// TwinCAT 3 PLC project PLC3
// ProgramVersion: 3.1.4022.3
// libraries:
//   Tc2_Standard, * (Beckhoff Automation GmbH)
//   Tc2_System, * (Beckhoff Automation GmbH)
//   Tc3_Module, * (Beckhoff Automation GmbH)
// project tree:
//   DUTs/ Drinks.TcDUT (not stored), States.TcDUT (not stored)
//   / GlobalTextList.TcGTLO (not stored), PlcTask.TcTTO (not stored), Visualization Manager.TcVMO (not stored)
//   GVLs/ GVL_IO.TcGVL
//   POUs/ FindFree.TcPOU, MAIN.TcPOU, MoveArm.TcPOU, CountFreeSpaces.TcPOU (not stored)
// real-time tasks:
//   TASK PlcTask: cycle T#10ms, priority 20, ADS port 350
// I/O:
//   DEVICE Device 1 (EtherCAT), AmsNetId 5.17.58.102.2.1
//     Term 1 (EK1200) [EK1200-5000 EtherCAT Power supply (2A E-Bus)]
//       Term 2 (EK1110) [EK1110 EtherCAT extension]
//     Term 3 (EK1100) [EK1100 EtherCAT Coupler (2A E-Bus)]
//       Term 4 (EL1809) [EL1809 16Ch. Dig. Input 24V, 3ms]
//       Term 5 (EL1809) [EL1809 16Ch. Dig. Input 24V, 3ms]
//       Term 6 (EL2809) [EL2809 16Ch. Dig. Output 24V, 0.5A]
//       Term 7 (EL2809) [EL2809 16Ch. Dig. Output 24V, 0.5A]
//       Term 8 (EL9011) [EL9011 End Terminal]
//   DEVICE Device 2 (EtherCAT Automation Protocol) (disabled), AmsNetId 5.17.58.102.3.1
//   DEVICE Device 5 (RT-Ethernet Protocol) (disabled), AmsNetId 5.17.58.102.6.1
// variable links:
//   PLC3/PLC3 Instance <-> Device 1 (EtherCAT)/Term 3 (EK1100)/Term 4 (EL1809)
//     PlcTask Inputs/GVL_IO.ALARMX_ALARM_tableX <-> Channel 11/Input
//     PlcTask Inputs/GVL_IO.ALARMY_ALARM_translationY <-> Channel 15/Input
//     PlcTask Inputs/GVL_IO.Auto_I_Manual_II_switch <-> Channel 3/Input
//     PlcTask Inputs/GVL_IO.BUSYX_BUSY_tableX <-> Channel 9/Input
//     PlcTask Inputs/GVL_IO.BUSYY_BUSY_traslationY <-> Channel 13/Input
//     PlcTask Inputs/GVL_IO.EMERX_EMERGENCY_tableX <-> Channel 12/Input
//     PlcTask Inputs/GVL_IO.EMERY_EMERGENCY_translationY <-> Channel 16/Input
//     PlcTask Inputs/GVL_IO.Reset_button <-> Channel 4/Input
//     PlcTask Inputs/GVL_IO.SETONX_ORIGIN_tableX <-> Channel 10/Input
//     PlcTask Inputs/GVL_IO.SETONY_ORIGIN_translationY <-> Channel 14/Input
//     PlcTask Inputs/GVL_IO.Start_button <-> Channel 1/Input
//     PlcTask Inputs/GVL_IO.Stop_button <-> Channel 2/Input
//     PlcTask Inputs/GVL_IO.a_0_Vertical_Zaxis_upward <-> Channel 5/Input
//     PlcTask Inputs/GVL_IO.a_1_Vertical_Zaxis_downward <-> Channel 6/Input
//     PlcTask Inputs/GVL_IO.dp1_Can_detection <-> Channel 7/Input
//     PlcTask Inputs/GVL_IO.dp2_Cover_detection <-> Channel 8/Input
//   PLC3/PLC3 Instance <-> Device 1 (EtherCAT)/Term 3 (EK1100)/Term 6 (EL2809)
//     PlcTask Outputs/GVL_IO.Aplus_Vert_axis_downwards <-> Channel 2/Output
//     PlcTask Outputs/GVL_IO.BR_Alarm_light <-> Channel 1/Output
//     PlcTask Outputs/GVL_IO.DRIVEX_MOVE_tableX <-> Channel 10/Output
//     PlcTask Outputs/GVL_IO.DRIVEY_MOVE_translY <-> Channel 16/Output
//     PlcTask Outputs/GVL_IO.HOLD_STOP_tableX_AND_translY <-> Channel 9/Output
//     PlcTask Outputs/GVL_IO.INX0_from_Input0_tableX <-> Channel 4/Output
//     PlcTask Outputs/GVL_IO.INX1_from_Input1_tableX <-> Channel 5/Output
//     PlcTask Outputs/GVL_IO.INX2_from_Input2_tableX <-> Channel 6/Output
//     PlcTask Outputs/GVL_IO.INY0_from_Input0_translY <-> Channel 11/Output
//     PlcTask Outputs/GVL_IO.INY1_from_Input1_translY <-> Channel 12/Output
//     PlcTask Outputs/GVL_IO.INY2_from_Input2_translY <-> Channel 13/Output
//     PlcTask Outputs/GVL_IO.SETUPX_ORIGIN_tableX <-> Channel 8/Output
//     PlcTask Outputs/GVL_IO.SETUPY_ORIGIN_translY <-> Channel 15/Output
//     PlcTask Outputs/GVL_IO.SVONX_SERVO_ON_tableX <-> Channel 7/Output
//     PlcTask Outputs/GVL_IO.SVONY_SERVO_ON_translY <-> Channel 14/Output
//     PlcTask Outputs/GVL_IO.Vplus_Vacuum_start <-> Channel 3/Output

// ---- GVLs/GVL_IO.TcGVL
{attribute 'qualified_only'}     // Do not remove this line
VAR_GLOBAL
// Input module EL1809	
    Start_button                 AT %I* :BOOL;
    Stop_button                  AT %I* :BOOL;
    Auto_I_Manual_II_switch      AT %I* :BOOL;
    Reset_button                 AT %I* :BOOL;
    a_0_Vertical_Zaxis_upward    AT %I* :BOOL;
    a_1_Vertical_Zaxis_downward  AT %I* :BOOL;
    dp1_Can_detection            AT %I* :BOOL;
    dp2_Cover_detection          AT %I* :BOOL;
    BUSYX_BUSY_tableX            AT %I* :BOOL;
    SETONX_ORIGIN_tableX         AT %I* :BOOL;
    ALARMX_ALARM_tableX          AT %I* :BOOL;
    EMERX_EMERGENCY_tableX       AT %I* :BOOL;
    BUSYY_BUSY_traslationY       AT %I* :BOOL;
    SETONY_ORIGIN_translationY   AT %I* :BOOL;
    ALARMY_ALARM_translationY    AT %I* :BOOL;
    EMERY_EMERGENCY_translationY AT %I* :BOOL;
//========================================
	INPUTchannel_01_SPARE        AT %I* :BOOL;
	INPUTchannel_02_SPARE        AT %I* :BOOL;
	INPUTchannel_03_SPARE        AT %I* :BOOL;
	INPUTchannel_04_SPARE        AT %I* :BOOL;
	INPUTchannel_05_SPARE        AT %I* :BOOL;
	INPUTchannel_06_SPARE        AT %I* :BOOL;
	INPUTchannel_07_SPARE        AT %I* :BOOL;
	INPUTchannel_08_SPARE        AT %I* :BOOL;
	INPUTchannel_09_SPARE        AT %I* :BOOL;
	INPUTchannel_10_SPARE        AT %I* :BOOL;
	INPUTchannel_11_SPARE        AT %I* :BOOL;
	INPUTchannel_12_SPARE        AT %I* :BOOL;
	INPUTchannel_13_SPARE        AT %I* :BOOL;
	INPUTchannel_14_SPARE        AT %I* :BOOL;
	INPUTchannel_15_SPARE        AT %I* :BOOL;
	INPUTchannel_16_SPARE        AT %I* :BOOL;
//========================================
	BR_Alarm_light               AT %Q* :BOOL;
    Aplus_Vert_axis_downwards    AT %Q* :BOOL;
    Vplus_Vacuum_start           AT %Q* :BOOL;
    INX0_from_Input0_tableX      AT %Q* :BOOL;
    INX1_from_Input1_tableX      AT %Q* :BOOL;
    INX2_from_Input2_tableX      AT %Q* :BOOL;
    SVONX_SERVO_ON_tableX        AT %Q* :BOOL;
    SETUPX_ORIGIN_tableX         AT %Q* :BOOL;
    HOLD_STOP_tableX_AND_translY AT %Q* :BOOL;
    DRIVEX_MOVE_tableX           AT %Q* :BOOL;
    INY0_from_Input0_translY     AT %Q* :BOOL;
    INY1_from_Input1_translY     AT %Q* :BOOL;
    INY2_from_Input2_translY     AT %Q* :BOOL;
    SVONY_SERVO_ON_translY       AT %Q* :BOOL;
    SETUPY_ORIGIN_translY        AT %Q* :BOOL;
    DRIVEY_MOVE_translY          AT %Q* :BOOL;
//============================================
    OUTPUTchannel_01_SPARE       AT %Q* :BOOL;
    OUTPUTchannel_02_SPARE       AT %Q* :BOOL;
    OUTPUTchannel_03_SPARE       AT %Q* :BOOL;
    OUTPUTchannel_04_SPARE       AT %Q* :BOOL;
    OUTPUTchannel_05_SPARE       AT %Q* :BOOL;
    OUTPUTchannel_06_SPARE       AT %Q* :BOOL;
    OUTPUTchannel_07_SPARE       AT %Q* :BOOL;
    OUTPUTchannel_08_SPARE       AT %Q* :BOOL;
    OUTPUTchannel_00_SPARE       AT %Q* :BOOL;
    OUTPUTchannel_10_SPARE       AT %Q* :BOOL;
    OUTPUTchannel_11_SPARE       AT %Q* :BOOL;
    OUTPUTchannel_12_SPARE       AT %Q* :BOOL;
    OUTPUTchannel_13_SPARE       AT %Q* :BOOL;
    OUTPUTchannel_14_SPARE       AT %Q* :BOOL;
    OUTPUTchannel_15_SPARE       AT %Q* :BOOL;
    OUTPUTchannel_16_SPARE       AT %Q* :BOOL;
END_VAR

// ---- POUs/FindFree.TcPOU
FUNCTION_BLOCK FindFree
VAR_INPUT
	DrinkArray: ARRAY [1..25] OF Drinks;
	PalletArray: ARRAY [1..25] OF BOOL;
	TempDrink : Drinks;
END_VAR
VAR_OUTPUT
	FreePosition : INT; 
END_VAR
VAR
	Counter : INT;
END_VAR

FreePosition := 666;

FOR Counter:=1 TO 25 DO //sizeof array werkt niet
 	IF NOT PalletArray[Counter] THEN
		IF DrinkArray[Counter] = TempDrink THEN
		FreePosition := Counter;
		END_IF
	END_IF
END_FOR
// counter gaat van 25 naar 1 ipv 1 naar 25... onzin.
// fanta plaatsen worden niet gezien, cola komt er alsnog op

END_FUNCTION_BLOCK

// ---- POUs/MAIN.TcPOU
PROGRAM MAIN
VAR
	Timer1 :TON;
	Timer2 : TON;
	PulseTimer1 : TP;

	CurrentState  : States;
	
	ServoRTrigY : R_Trig ; 
	ServoRTrigX : R_Trig ; 
	
	//Eigen trigger booleans
	InitYReady : BOOL;
	InitXReady : BOOL;
	droppingDown : BOOL; //test
	
	TimerTest1 : TIME;
	TimerResult : TIME;
	
	Move_Arm : MoveArm;
	Count_Free_Spaces : CountFreeSpaces;
	Find_Free : FindFree;
	
	PalletArray: ARRAY [1..25] OF BOOL := [25(FALSE)];
	
	DrinkArray: ARRAY [1..25] OF Drinks := [13(Drinks.Cola), 12(Drinks.Fanta)]; 
	FreeCola : INT;
	FreeFanta : INT;
	
	//messages voor Nicky & Jens
	BottleAvailable : BOOL;
	CorrectDelivery : BOOL;
	NoCover : BOOL;
	NoBottle : BOOL;
	WrongDrink : BOOL;
	ColaFanta: INT;
	
	//Settings
	StartPos : INT;
	ErrorPos: INT;
	CurrentPos : INT;
	
	
END_VAR

PulseTimer1(IN:=GVL_IO.Start_button, PT:=T#150MS);
Timer1(IN:= GVL_IO.a_1_Vertical_Zaxis_downward, PT:= T#10MS);
Timer2(IN:=droppingDown AND NOT GVL_IO.a_1_Vertical_Zaxis_downward, PT:=T#280MS);

CASE CurrentState OF
States.Init:
		//Aanzetten van servo's. Dit kan even duren GEEN HOMING
		GVL_IO.SVONX_SERVO_ON_tableX 	  := TRUE; 
		GVL_IO.SVONY_SERVO_ON_translY 	  := TRUE;
		
		GVL_IO.SETUPX_ORIGIN_tableX := PulseTimer1.Q;
		GVL_IO.SETUPY_ORIGIN_translY := PulseTimer1.Q;
		
		//// Koppelen van outputs Busy aan var's. Triggered op een falling edge.
		IF PulseTimer1.Q THEN
			ServoRTrigX ( clk := gvl_io.SETONX_ORIGIN_tableX ); 
	  		ServoRTrigY ( clk := gvl_io.SETONY_ORIGIN_translationY );
		END_IF
		
		// Bools setten aan de hand van triggers.
		IF ServoRTrigX.Q THEN
			InitXReady:= TRUE;
		END_IF
		
		IF ServoRTrigY.Q THEN
			InitYReady:= TRUE;
		END_IF
		
		// Init voltooid ga naar idle
		IF InitXReady AND InitYReady THEN
			CurrentPos:= 1;
			NoCover := FALSE;
			NoBottle := FALSE;
			WrongDrink:= FALSE;
			CorrectDelivery := FALSE;
			ErrorPos:= 666;
			StartPos:= 30;
			ColaFanta := drinks.Cola;
			CurrentState:= States.Idle;
		END_IF
		
States.Idle:
		//=========================TEST=================================
		IF NOT GVL_IO.Stop_button THEN
			BottleAvailable := TRUE;
		END_IF
		//==============================================================
		CorrectDelivery := FALSE;
		Count_Free_Spaces(DrinkArray:=DrinkArray, PalletArray:= PalletArray);
		FreeCola := Count_Free_Spaces.FreeCola;
		FreeFanta := Count_Free_Spaces.FreeFanta;
		IF BottleAvailable AND GVL_IO.dp1_Can_detection AND GVL_IO.dp2_Cover_detection THEN
			Find_Free(DrinkArray:=DrinkArray, PalletArray:= PalletArray, TempDrink:= ColaFanta, ErrorPosition:=ErrorPos);
			CurrentPos := Find_Free.FreePosition;
			IF CurrentPos = ErrorPos THEN
				WrongDrink := TRUE;
				CurrentState := States.ManualCheck;
			ELSE
				CorrectDelivery := TRUE;
				NoCover := FALSE;
				NoBottle := FALSE;
				CurrentState := States.MoveToPickUp;
			END_IF
		ELSIF BottleAvailable AND NOT GVL_IO.dp1_Can_detection THEN
			NoBottle := TRUE;
		ELSIF BottleAvailable AND NOT GVL_IO.dp2_Cover_detection THEN
			NoCover := TRUE;
		END_IF
		BottleAvailable := FALSE;
		
States.MoveToPickUp:
		Move_Arm(Position:= StartPos);
		IF Move_Arm.OnNewLocation THEN
			CurrentState := States.PickUpDown;
		END_IF
		
States.PickUpDown:
		IF GVL_IO.a_0_Vertical_Zaxis_upward THEN
			GVL_IO.Aplus_Vert_axis_downwards := TRUE;
		END_IF
		
		IF GVL_IO.a_1_Vertical_Zaxis_downward THEN
			GVL_IO.Vplus_Vacuum_start := TRUE;
			
			IF Timer1.Q THEN
			CurrentState := States.PickUpUp;
			END_IF
		END_IF

States.PickUpUp:
		GVL_IO.Aplus_Vert_axis_downwards := FALSE;
		
		IF GVL_IO.a_0_Vertical_Zaxis_upward THEN
			CurrentState := States.Moving;
		END_IF
		
States.Moving:
		IF GVL_IO.a_0_Vertical_Zaxis_upward THEN
			Move_Arm(Position:= CurrentPos);
			IF Move_Arm.OnNewLocation THEN
				PalletArray[CurrentPos] := TRUE;
				CurrentState := States.DropDown;
			END_IF
		END_IF
		
States.DropDown:
		IF GVL_IO.a_0_Vertical_Zaxis_upward THEN
			GVL_IO.Aplus_Vert_axis_downwards := TRUE;
			droppingDown := TRUE;
			TimerTest1 := TIME();
		END_IF
		
		
		IF 	GVL_IO.a_1_Vertical_Zaxis_downward THEN
			GVL_IO.Vplus_Vacuum_start := FALSE;
			IF Timer1.Q THEN
				TimerResult := TIME() - TimerTest1;
				droppingDown := FALSE;
				CurrentState := States.DropUp;
			END_IF
			
		ELSE IF Timer2.Q  THEN
		GVL_io.Aplus_Vert_axis_downwards := FALSE;
		droppingDown := FALSE;
		CurrentState := States.ManualCheck;
		END_IF
		END_IF

States.DropUp:
		IF GVL_IO.a_1_Vertical_Zaxis_downward THEN
			GVL_IO.Aplus_Vert_axis_downwards := FALSE;
		END_IF
		
		IF GVL_IO.a_0_Vertical_Zaxis_upward THEN
			//BottleAvailable := FALSE;
			CurrentState := States.Idle;
		END_IF
		
States.ManualCheck:
		GVL_IO.BR_Alarm_light := TRUE;
		GVL_io.Vplus_Vacuum_start := FALSE;
		IF GVL_IO.Reset_button THEN
			GVL_IO.BR_Alarm_light := FALSE;
			WrongDrink := FALSE;
			Currentstate := States.Idle;
		END_IF
END_CASE

END_PROGRAM

// ---- POUs/MoveArm.TcPOU
FUNCTION_BLOCK MoveArm
VAR_INPUT
Position: INT;
END_VAR
VAR_OUTPUT
	OnNewLocation:BOOL;
END_VAR
VAR
	X: INT;
	Y: INT;
	StartTimer:BOOL;
	
	PulseTimer2: TP;
	BusyFtrigX : F_Trig;
	BusyFtrigY : F_Trig;
	ReadyX : BOOL;
	ReadyY : BOOL;
	Busy: BOOL;
END_VAR

OnNewLocation := FALSE;

IF( Position < 1 OR Position > 30)  
	THEN RETURN; 
END_IF

// Calculate X & Y position on Palletiser
// 
X := (Position - 1) MOD 5;

// Position-1 / 5 with ROUND to floor 
Y := ((Position -1) / 5) - ((Position -1) / 5) MOD 1;

// set position 
GVL_IO.INX0_from_Input0_tableX:= X.0;
GVL_IO.INX1_from_Input1_tableX:= X.1;
GVL_IO.INX2_from_Input2_tableX:= X.2;
GVL_IO.INY0_from_Input0_translY:= Y.0;
GVL_IO.INY1_from_Input1_translY:= Y.1;
GVL_IO.INY2_from_Input2_translY:= Y.2;



PulseTimer2(IN:=StartTimer, PT:=T#150MS);

GVL_IO.DRIVEX_MOVE_tableX := PulseTimer2.Q;
GVL_IO.DRIVEY_MOVE_translY := PulseTimer2.Q;
StartTimer:= TRUE;
		
BusyFtrigX ( clk := gvl_io.BUSYX_BUSY_tableX ); 
BusyFtrigY ( clk := gvl_io.BUSYY_BUSY_traslationY );
		
IF BusyFtrigX.Q THEN
	ReadyX:= TRUE;
END_IF
		
IF BusyFtrigY.Q THEN
	ReadyY:= TRUE;
END_IF
		
IF ReadyY AND ReadyX THEN
	GVL_IO.DRIVEX_MOVE_tableX := FALSE;
	GVL_IO.DRIVEY_MOVE_translY := FALSE;
	ReadyX:= FALSE;
	ReadyY:= FALSE;
	StartTimer:= FALSE;
	OnNewLocation := TRUE;
END_IF

END_FUNCTION_BLOCK
